(* IEC 61131-3 sources: SafePLC-Gen-Evaluation/Evaluation Results/dexpi/run_05, 2 files *)

(* ---- io_declarations.st ---- *)
(* ==================================================  *)
(* PLC I/O Variable Declarations — CODESYS 3.5  *)
(* Generated by SafePLC-Gen Multimodal  *)
(* ==================================================  *)

VAR_GLOBAL
    (* --- Analog Inputs ---  *)
    PI_4712.01_Raw               AT %IW0       : INT := 0;    (* PI-4712.01 — Pressure indicator (local gauge) on disc  *)
    PICSA_4712.02_Raw            AT %IW2       : INT := 0;    (* PICSA-4712.02 — Pressure Indicator, Controller, Switch w  *)
    TICSA_4750.03_Raw            AT %IW4       : INT := 0;    (* TICSA-4750.03 — Temperature Indicator, Controller, Switc  *)
    (* --- Analog Outputs ---  *)
    PV_4712.02_Out               AT %QW0       : INT := 0;    (* PV-4712.02 — Pressure control valve, globe body with   *)
    TV_4750.03_Out               AT %QW2       : INT := 0;    (* TV-4750.03 — Temperature control valve, globe body wi  *)
    (* --- Digital Inputs ---  *)
    HS_4750.01                   AT %IX0.0     : BOOL := FALSE;    (* HS-4750.01 — Hand switch (operator pushbutton/selecto  *)
    (* --- Digital Outputs ---  *)
    XV_4750.01                   AT %QX0.0     : BOOL := FALSE;    (* XV-4750.01 — Solenoid-operated on/off valve on T4750   *)
END_VAR

(* ---- generated_code.st ---- *)
(* Generated by SafePLC-Gen Multimodal — CODESYS 3.5 *)
(* IEC 61131-3 Structured Text *)
(* Date: 2026-04-25T11:54:49.826380 *)

PROGRAM PressureTemperatureControl

VAR
    TICSA_4750_03_Raw            AT %IW4       : INT := 0;
    PICSA_4712_02_Raw            AT %IW2       : INT := 0;
    PI_4712_01_Raw               AT %IW0       : INT := 0;
    HS_4750_01                   AT %IX0.0     : BOOL := FALSE;
    PV_4712_02_Out               AT %QW0       : INT := 0;
    TV_4750_03_Out               AT %QW2       : INT := 0;
    XV_4750_01                   AT %QX0.0     : BOOL := FALSE;
    ESTOP                        AT %IX0.1     : BOOL := FALSE;
    MANUAL_RESET                 AT %IX0.2     : BOOL := FALSE;
END_VAR

VAR
    FirstScan                    : BOOL := TRUE;

    TICSA_4750_03_Scaled         : REAL := 0.0;
    PICSA_4712_02_Scaled         : REAL := 0.0;
    PI_4712_01_Scaled            : REAL := 0.0;

    TICSA_4750_03_EU_Min         : REAL := 0.0;
    TICSA_4750_03_EU_Span        : REAL := 200.0;
    PICSA_4712_02_EU_Min         : REAL := 0.0;
    PICSA_4712_02_EU_Span        : REAL := 100.0;
    PI_4712_01_EU_Min            : REAL := 0.0;
    PI_4712_01_EU_Span           : REAL := 100.0;

    TICSA_4750_03_HH_SP          : REAL := 180.0;
    TICSA_4750_03_H_SP           : REAL := 160.0;
    TICSA_4750_03_L_SP           : REAL := 20.0;
    TICSA_4750_03_LL_SP          : REAL := 10.0;
    TICSA_4750_03_Deadband       : REAL := 2.0;

    PICSA_4712_02_HH_SP          : REAL := 90.0;
    PICSA_4712_02_H_SP           : REAL := 80.0;
    PICSA_4712_02_L_SP           : REAL := 10.0;
    PICSA_4712_02_LL_SP          : REAL := 5.0;
    PICSA_4712_02_Deadband       : REAL := 1.0;

    PI_4712_01_HH_SP             : REAL := 90.0;
    PI_4712_01_H_SP              : REAL := 80.0;
    PI_4712_01_L_SP              : REAL := 10.0;
    PI_4712_01_LL_SP             : REAL := 5.0;
    PI_4712_01_Deadband          : REAL := 1.0;

    TICSA_4750_03_HH_Ack         : BOOL := FALSE;
    TICSA_4750_03_LL_Ack         : BOOL := FALSE;
    PICSA_4712_02_HH_Ack         : BOOL := FALSE;
    PICSA_4712_02_LL_Ack         : BOOL := FALSE;
    PI_4712_01_HH_Ack            : BOOL := FALSE;
    PI_4712_01_LL_Ack            : BOOL := FALSE;

    (* HH/LL latched alarm states — set by alarm logic, cleared by ack+normal *)
    TICSA_4750_03_HH_Latched     : BOOL := FALSE;
    TICSA_4750_03_LL_Latched     : BOOL := FALSE;
    PICSA_4712_02_HH_Latched     : BOOL := FALSE;
    PICSA_4712_02_LL_Latched     : BOOL := FALSE;
    PI_4712_01_HH_Latched        : BOOL := FALSE;
    PI_4712_01_LL_Latched        : BOOL := FALSE;

    TICSA_4750_03_HH             : BOOL := FALSE;
    TICSA_4750_03_LL             : BOOL := FALSE;
    TICSA_4750_03_H              : BOOL := FALSE;
    TICSA_4750_03_L              : BOOL := FALSE;

    PICSA_4712_02_HH             : BOOL := FALSE;
    PICSA_4712_02_LL             : BOOL := FALSE;
    PICSA_4712_02_H              : BOOL := FALSE;
    PICSA_4712_02_L              : BOOL := FALSE;

    PI_4712_01_HH                : BOOL := FALSE;
    PI_4712_01_LL                : BOOL := FALSE;
    PI_4712_01_H                 : BOOL := FALSE;
    PI_4712_01_L                 : BOOL := FALSE;

    LOOP_4750_03_TRIP            : BOOL := FALSE;
    LOOP_4712_02_TRIP            : BOOL := FALSE;
    LOOP_104_01_TRIP             : BOOL := FALSE;
    SV_104_01_HH                 : BOOL := FALSE;
    SV_104_01_LL                 : BOOL := FALSE;
    SAFE_STATE                   : BOOL := FALSE;

    TIC_SP                       : REAL := 80.0;
    TIC_Error                    : REAL := 0.0;
    TIC_Integral                 : REAL := 50.0;
    TIC_Kp                       : REAL := 2.0;
    TIC_Ki                       : REAL := 0.05;
    TIC_Output                   : REAL := 0.0;

    PIC_SP                       : REAL := 50.0;
    PIC_Error                    : REAL := 0.0;
    PIC_Integral                 : REAL := 50.0;
    PIC_Kp                       : REAL := 2.0;
    PIC_Ki                       : REAL := 0.05;
    PIC_Output                   : REAL := 0.0;

    HV_MNb_47121                 : BOOL := FALSE;
    HV_MNb_47122                 : BOOL := FALSE;
    HV_75SA21                    : BOOL := FALSE;
    CV_73KH12_50_inlet           : BOOL := FALSE;
    HV_MNc_47125_block           : BOOL := FALSE;
    HV_MNc_47126                 : BOOL := FALSE;
    HV_73KH12_50_main            : BOOL := FALSE;
    HV_QSa_47140                 : BOOL := FALSE;
    HV_QSb_47141                 : BOOL := FALSE;
    HV_MNc_47127_Q80             : BOOL := FALSE;
    HV_66KL21                    : BOOL := FALSE;
    HV_73KH12_25_PI              : BOOL := FALSE;
    HV_73KH12_25_PICSA           : BOOL := FALSE;
    SV_104_01_Out                : BOOL := FALSE;

    System_Alarm                 : BOOL := FALSE;
END_VAR

IF FirstScan THEN
    LOOP_4750_03_TRIP    := TRUE;
    LOOP_4712_02_TRIP    := TRUE;
    LOOP_104_01_TRIP     := TRUE;
    SAFE_STATE           := TRUE;
    TV_4750_03_Out       := 6554;
    PV_4712_02_Out       := 6554;
    XV_4750_01           := FALSE;
    SV_104_01_Out        := FALSE;
    HV_MNb_47121         := FALSE;
    HV_MNb_47122         := FALSE;
    HV_75SA21            := FALSE;
    CV_73KH12_50_inlet   := FALSE;
    HV_MNc_47125_block   := FALSE;
    HV_MNc_47126         := FALSE;
    HV_73KH12_50_main    := FALSE;
    HV_QSa_47140         := FALSE;
    HV_QSb_47141         := FALSE;
    HV_MNc_47127_Q80     := FALSE;
    HV_66KL21            := FALSE;
    HV_73KH12_25_PI      := FALSE;
    HV_73KH12_25_PICSA   := FALSE;
    TIC_Integral         := 50.0;
    PIC_Integral         := 50.0;
    TICSA_4750_03_HH_Latched := FALSE;
    TICSA_4750_03_LL_Latched := FALSE;
    PICSA_4712_02_HH_Latched := FALSE;
    PICSA_4712_02_LL_Latched := FALSE;
    PI_4712_01_HH_Latched    := FALSE;
    PI_4712_01_LL_Latched    := FALSE;
    FirstScan            := FALSE;
    RETURN;
END_IF;

TICSA_4750_03_Scaled := ((INT_TO_REAL(TICSA_4750_03_Raw) - 6554.0) / (32767.0 - 6554.0)) * TICSA_4750_03_EU_Span + TICSA_4750_03_EU_Min;
PICSA_4712_02_Scaled := ((INT_TO_REAL(PICSA_4712_02_Raw) - 6554.0) / (32767.0 - 6554.0)) * PICSA_4712_02_EU_Span + PICSA_4712_02_EU_Min;
PI_4712_01_Scaled    := ((INT_TO_REAL(PI_4712_01_Raw)    - 6554.0) / (32767.0 - 6554.0)) * PI_4712_01_EU_Span    + PI_4712_01_EU_Min;

(* TICSA-4750.03 HH latching alarm *)
IF TICSA_4750_03_Scaled >= TICSA_4750_03_HH_SP THEN
    TICSA_4750_03_HH_Latched := TRUE;
ELSIF TICSA_4750_03_HH_Ack AND (TICSA_4750_03_Scaled <= (TICSA_4750_03_HH_SP - TICSA_4750_03_Deadband)) THEN
    TICSA_4750_03_HH_Latched := FALSE;
END_IF;
TICSA_4750_03_HH := TICSA_4750_03_HH_Latched;

(* TICSA-4750.03 LL latching alarm *)
IF TICSA_4750_03_Scaled <= TICSA_4750_03_LL_SP THEN
    TICSA_4750_03_LL_Latched := TRUE;
ELSIF TICSA_4750_03_LL_Ack AND (TICSA_4750_03_Scaled >= (TICSA_4750_03_LL_SP + TICSA_4750_03_Deadband)) THEN
    TICSA_4750_03_LL_Latched := FALSE;
END_IF;
TICSA_4750_03_LL := TICSA_4750_03_LL_Latched;

(* TICSA-4750.03 H/L non-latching *)
IF TICSA_4750_03_Scaled >= TICSA_4750_03_H_SP THEN
    TICSA_4750_03_H := TRUE;
ELSIF TICSA_4750_03_Scaled <= (TICSA_4750_03_H_SP - TICSA_4750_03_Deadband) THEN
    TICSA_4750_03_H := FALSE;
END_IF;

IF TICSA_4750_03_Scaled <= TICSA_4750_03_L_SP THEN
    TICSA_4750_03_L := TRUE;
ELSIF TICSA_4750_03_Scaled >= (TICSA_4750_03_L_SP + TICSA_4750_03_Deadband) THEN
    TICSA_4750_03_L := FALSE;
END_IF;

(* PICSA-4712.02 HH latching alarm *)
IF PICSA_4712_02_Scaled >= PICSA_4712_02_HH_SP THEN
    PICSA_4712_02_HH_Latched := TRUE;
ELSIF PICSA_4712_02_HH_Ack AND (PICSA_4712_02_Scaled <= (PICSA_4712_02_HH_SP - PICSA_4712_02_Deadband)) THEN
    PICSA_4712_02_HH_Latched := FALSE;
END_IF;
PICSA_4712_02_HH := PICSA_4712_02_HH_Latched;

(* PICSA-4712.02 LL latching alarm *)
IF PICSA_4712_02_Scaled <= PICSA_4712_02_LL_SP THEN
    PICSA_4712_02_LL_Latched := TRUE;
ELSIF PICSA_4712_02_LL_Ack AND (PICSA_4712_02_Scaled >= (PICSA_4712_02_LL_SP + PICSA_4712_02_Deadband)) THEN
    PICSA_4712_02_LL_Latched := FALSE;
END_IF;
PICSA_4712_02_LL := PICSA_4712_02_LL_Latched;

(* PICSA-4712.02 H/L non-latching *)
IF PICSA_4712_02_Scaled >= PICSA_4712_02_H_SP THEN
    PICSA_4712_02_H := TRUE;
ELSIF PICSA_4712_02_Scaled <= (PICSA_4712_02_H_SP - PICSA_4712_02_Deadband) THEN
    PICSA_4712_02_H := FALSE;
END_IF;

IF PICSA_4712_02_Scaled <= PICSA_4712_02_L_SP THEN
    PICSA_4712_02_L := TRUE;
ELSIF PICSA_4712_02_Scaled >= (PICSA_4712_02_L_SP + PICSA_4712_02_Deadband) THEN
    PICSA_4712_02_L := FALSE;
END_IF;

(* PI-4712.01 HH latching alarm *)
IF PI_4712_01_Scaled >= PI_4712_01_HH_SP THEN
    PI_4712_01_HH_Latched := TRUE;
ELSIF PI_4712_01_HH_Ack AND (PI_4712_01_Scaled <= (PI_4712_01_HH_SP - PI_4712_01_Deadband)) THEN
    PI_4712_01_HH_Latched := FALSE;
END_IF;
PI_4712_01_HH := PI_4712_01_HH_Latched;

(* PI-4712.01 LL latching alarm *)
IF PI_4712_01_Scaled <= PI_4712_01_LL_SP THEN
    PI_4712_01_LL_Latched := TRUE;
ELSIF PI_4712_01_LL_Ack AND (PI_4712_01_Scaled >= (PI_4712_01_LL_SP + PI_4712_01_Deadband)) THEN
    PI_4712_01_LL_Latched := FALSE;
END_IF;
PI_4712_01_LL := PI_4712_01_LL_Latched;

(* PI-4712.01 H/L non-latching *)
IF PI_4712_01_Scaled >= PI_4712_01_H_SP THEN
    PI_4712_01_H := TRUE;
ELSIF PI_4712_01_Scaled <= (PI_4712_01_H_SP - PI_4712_01_Deadband) THEN
    PI_4712_01_H := FALSE;
END_IF;

IF PI_4712_01_Scaled <= PI_4712_01_L_SP THEN
    PI_4712_01_L := TRUE;
ELSIF PI_4712_01_Scaled >= (PI_4712_01_L_SP + PI_4712_01_Deadband) THEN
    PI_4712_01_L := FALSE;
END_IF;

(* Safety trip latches *)
IF TICSA_4750_03_HH OR TICSA_4750_03_LL THEN
    LOOP_4750_03_TRIP := TRUE;
ELSIF LOOP_4750_03_TRIP AND MANUAL_RESET AND NOT TICSA_4750_03_HH AND NOT TICSA_4750_03_LL THEN
    LOOP_4750_03_TRIP := FALSE;
END_IF;

IF PICSA_4712_02_HH OR PICSA_4712_02_LL THEN
    LOOP_4712_02_TRIP := TRUE;
ELSIF LOOP_4712_02_TRIP AND MANUAL_RESET AND NOT PICSA_4712_02_HH AND NOT PICSA_4712_02_LL THEN
    LOOP_4712_02_TRIP := FALSE;
END_IF;

IF SV_104_01_HH OR SV_104_01_LL THEN
    LOOP_104_01_TRIP := TRUE;
ELSIF LOOP_104_01_TRIP AND MANUAL_RESET AND NOT SV_104_01_HH AND NOT SV_104_01_LL THEN
    LOOP_104_01_TRIP := FALSE;
END_IF;

SAFE_STATE := ESTOP OR LOOP_4750_03_TRIP OR LOOP_4712_02_TRIP OR LOOP_104_01_TRIP;

IF NOT SAFE_STATE THEN
    TIC_Error    := TIC_SP - TICSA_4750_03_Scaled;
    TIC_Integral := TIC_Integral + (TIC_Ki * TIC_Error);
    IF TIC_Integral > 100.0 THEN
        TIC_Integral := 100.0;
    ELSIF TIC_Integral < 0.0 THEN
        TIC_Integral := 0.0;
    END_IF;
    TIC_Output := (TIC_Kp * TIC_Error) + TIC_Integral;
    IF TIC_Output > 100.0 THEN
        TIC_Output := 100.0;
    ELSIF TIC_Output < 0.0 THEN
        TIC_Output := 0.0;
    END_IF;
    TV_4750_03_Out := REAL_TO_INT(6554.0 + (TIC_Output / 100.0) * (32767.0 - 6554.0));

    PIC_Error    := PIC_SP - PICSA_4712_02_Scaled;
    PIC_Integral := PIC_Integral + (PIC_Ki * PIC_Error);
    IF PIC_Integral > 100.0 THEN
        PIC_Integral := 100.0;
    ELSIF PIC_Integral < 0.0 THEN
        PIC_Integral := 0.0;
    END_IF;
    PIC_Output := (PIC_Kp * PIC_Error) + PIC_Integral;
    IF PIC_Output > 100.0 THEN
        PIC_Output := 100.0;
    ELSIF PIC_Output < 0.0 THEN
        PIC_Output := 0.0;
    END_IF;
    PV_4712_02_Out := REAL_TO_INT(6554.0 + (PIC_Output / 100.0) * (32767.0 - 6554.0));

    XV_4750_01         := HS_4750_01;
    SV_104_01_Out      := TRUE;
    HV_MNb_47121       := TRUE;
    HV_MNb_47122       := TRUE;
    HV_75SA21          := TRUE;
    CV_73KH12_50_inlet := TRUE;
    HV_MNc_47125_block := TRUE;
    HV_MNc_47126       := TRUE;
    HV_73KH12_50_main  := TRUE;
    HV_QSa_47140       := TRUE;
    HV_QSb_47141       := TRUE;
    HV_MNc_47127_Q80   := TRUE;
    HV_66KL21          := TRUE;
    HV_73KH12_25_PI    := TRUE;
    HV_73KH12_25_PICSA := TRUE;
ELSE
    TV_4750_03_Out     := 6554;
    PV_4712_02_Out     := 6554;
    XV_4750_01         := FALSE;
    SV_104_01_Out      := FALSE;
    HV_MNb_47121       := FALSE;
    HV_MNb_47122       := FALSE;
    HV_75SA21          := FALSE;
    CV_73KH12_50_inlet := FALSE;
    HV_MNc_47125_block := FALSE;
    HV_MNc_47126       := FALSE;
    HV_73KH12_50_main  := FALSE;
    HV_QSa_47140       := FALSE;
    HV_QSb_47141       := FALSE;
    HV_MNc_47127_Q80   := FALSE;
    HV_66KL21          := FALSE;
    HV_73KH12_25_PI    := FALSE;
    HV_73KH12_25_PICSA := FALSE;
END_IF;

System_Alarm :=
    TICSA_4750_03_HH_Latched OR TICSA_4750_03_LL_Latched OR
    TICSA_4750_03_H          OR TICSA_4750_03_L          OR
    PICSA_4712_02_HH_Latched OR PICSA_4712_02_LL_Latched OR
    PICSA_4712_02_H          OR PICSA_4712_02_L          OR
    PI_4712_01_HH_Latched    OR PI_4712_01_LL_Latched    OR
    PI_4712_01_H             OR PI_4712_01_L             OR
    LOOP_4750_03_TRIP        OR LOOP_4712_02_TRIP        OR
    LOOP_104_01_TRIP         OR SAFE_STATE;

END_PROGRAM
